FUNCTION_BLOCK TaskManager (* Tamplate for a simple Basic Function Block Type *)
  (* Standard: 61499-2 *)
  (* Version 0.0, 2018-07-05, 4DIAC-IDE, 4DIAC-Consortium *)
  (* Version 1.0, 2016-05-26, AZ, fortiss GmbH *)
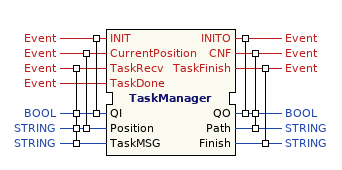
  EVENT_INPUT
    INIT WITH QI; (* Initialization Request *)
    CurrentPosition WITH Position;
    TaskRecv WITH QI, TaskMSG, Position; (* Normal Execution Request *)
    TaskDone;
  END_EVENT
  EVENT_OUTPUT
    INITO WITH QO; (* Initialization Confirm *)
    CNF WITH QO, Path; (* Execution Confirmation *)
    TaskFinish WITH Finish;
  END_EVENT
  VAR_INPUT
    QI : BOOL; (* Input event qualifier *)
    Position : STRING;
    TaskMSG : STRING; (* like 1_10 *)
  END_VAR
  VAR_OUTPUT
    QO : BOOL; (* Output event qualifier *)
    Path : STRING; (* like 1_10 *)
    Finish : STRING;
  END_VAR
  VAR
    TaskCount : INT := 0; (* Internal Variable *)
    Path1 : STRING; (* Internal Variable *)
    Paht2 : STRING; (* Internal Variable *)
  END_VAR
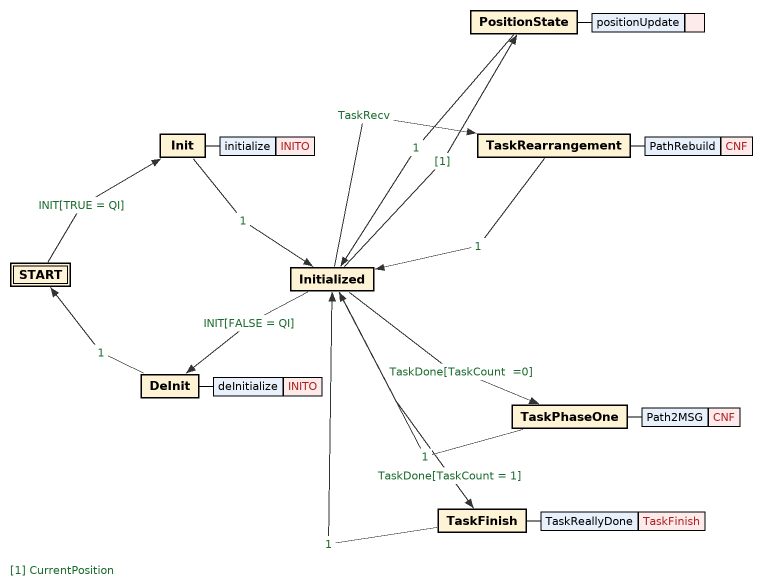
  EC_STATES
    START; (* Initial State *)
    Init : initialize -> INITO; (* Initialization *)
    TaskRearrangement : PathRebuild -> CNF; (* Normal execution *)
    Initialized;
    DeInit : deInitialize -> INITO;
    TaskPhaseOne : Path2MSG -> CNF;
    TaskFinish : TaskReallyDone -> TaskFinish;
    PositionState : positionUpdate;
  END_STATES
  EC_TRANSITIONS
    START TO Init := INIT[TRUE = QI];
    Init TO Initialized := 1;
    Initialized TO TaskRearrangement := TaskRecv;
    TaskRearrangement TO Initialized := 1;
    DeInit TO START := 1;
    Initialized TO DeInit := INIT[FALSE = QI];
    Initialized TO TaskPhaseOne := TaskDone[TaskCount  =0]; (* The first phase, AGV from initial position to task Begin position *)
    TaskPhaseOne TO Initialized := 1;
    Initialized TO TaskFinish := TaskDone[TaskCount = 1];
    TaskFinish TO Initialized := 1;
    Initialized TO PositionState := CurrentPosition;
    PositionState TO Initialized := 1;
  END_TRANSITIONS
  ALGORITHM initialize IN ST: (* Initialization algorithm *)
QO := QI;
  END_ALGORITHM
  ALGORITHM deInitialize IN ST: (* Normally executed algorithm *)
QO := FALSE;
  END_ALGORITHM
  ALGORITHM PathRebuild IN ST: (* new algorithm *)

  END_ALGORITHM
  ALGORITHM Path2MSG IN ST: (* new algorithm *)

  END_ALGORITHM
  ALGORITHM TaskReallyDone IN ST: (* new algorithm *)

  END_ALGORITHM
  ALGORITHM positionUpdate IN ST: (* new algorithm *)

  END_ALGORITHM
END_FUNCTION_BLOCK
